// TIA Portal project "final" (V16)

(* hardware
DEVICE "S7-1200 station_1"  S7-1200 Station
   slot 0: "Rack_0"  S7-1200 Rack  Rack  V1.0
   slot 1: "PLC_1"  CPU 1212C AC/DC/Rly  6ES7 212-1BE40-0XB0  V4.0
*)

// ===== PLC "PLC_1"  CPU 1212C AC/DC/Rly =====

VAR_GLOBAL   // PLC tag table "Default tag table"
   "Tag_1" AT %I0.7 : Bool;
   "Tag_2" AT %Q0.5 : Bool;
   "Tag_3" AT %M0.0 : Bool;
   "Tag_4" AT %M1.1 : Bool;
   "Tag_5" AT %M1.2 : Bool;
   "Tag_6" AT %M2.1 : Bool;
   "Tag_7" AT %Q0.3 : Bool;
   "Tag_8" AT %M0.1 : Bool;
   "Tag_9" AT %M1.3 : Bool;
   "Tag_10" AT %M3.1 : Bool;
   "Tag_11" AT %M0.2 : Bool;
   "Tag_12" AT %M4.1 : Bool;
   "Tag_13" AT %M3.2 : Bool;
   "Tag_14" AT %M2.2 : Bool;
   "Tag_15" AT %M0.3 : Bool;
   "Tag_16" AT %M4.2 : Bool;
   "Tag_17" AT %M3.3 : Bool;
   "Tag_18" AT %M2.3 : Bool;
   "Tag_19" AT %M0.5 : Bool;
   "Tag_20" AT %M4.3 : Bool;
   "Tag_21" AT %M0.6 : Bool;
   "Tag_22" AT %Q0.4 : Bool;
   "Tag_23" AT %Q0.2 : Bool;
END_VAR

// folder: System blocks/Program resources

DATA_BLOCK "0"   // DB1
{ S7_Optimized_Access := 'TRUE' }
AUTHOR : Simatic
FAMILY : IEC
NAME : IEC_TMR
VERSION : 1.0
// stored: InstanceOfName IEC_TIMER
"IEC_TIMER"
BEGIN
END_DATA_BLOCK

DATA_BLOCK "1"   // DB2
{ S7_Optimized_Access := 'TRUE' }
AUTHOR : Simatic
FAMILY : IEC
NAME : IEC_TMR
VERSION : 1.0
// stored: InstanceOfName IEC_TIMER
"IEC_TIMER"
BEGIN
END_DATA_BLOCK

DATA_BLOCK "2"   // DB3
{ S7_Optimized_Access := 'TRUE' }
AUTHOR : Simatic
FAMILY : IEC
NAME : IEC_TMR
VERSION : 1.0
// stored: InstanceOfName IEC_TIMER
"IEC_TIMER"
BEGIN
END_DATA_BLOCK

DATA_BLOCK "3"   // DB4
{ S7_Optimized_Access := 'TRUE' }
AUTHOR : Simatic
FAMILY : IEC
NAME : IEC_TMR
VERSION : 1.0
// stored: InstanceOfName IEC_TIMER
"IEC_TIMER"
BEGIN
END_DATA_BLOCK

DATA_BLOCK "4"   // DB5
{ S7_Optimized_Access := 'TRUE' }
AUTHOR : Simatic
FAMILY : IEC
NAME : IEC_TMR
VERSION : 1.0
// stored: InstanceOfName IEC_TIMER
"IEC_TIMER"
BEGIN
END_DATA_BLOCK

// folder: (top level)

ORGANIZATION_BLOCK "Main"   // OB1, LAD, ProgramCycle
TITLE = "Main Program Sweep (Cycle)"
{ S7_Optimized_Access := 'TRUE' }
VERSION : 0.1
   VAR_INPUT
      Initial_Call : Bool;   // Initial call of this OB
      Remanence : Bool;   // =True, if remanent data are available
   END_VAR
   VAR_TEMP   // added for the SCL form of the ladder/FBD networks
      _w1 : Bool;
   END_VAR
BEGIN

REGION Network 1
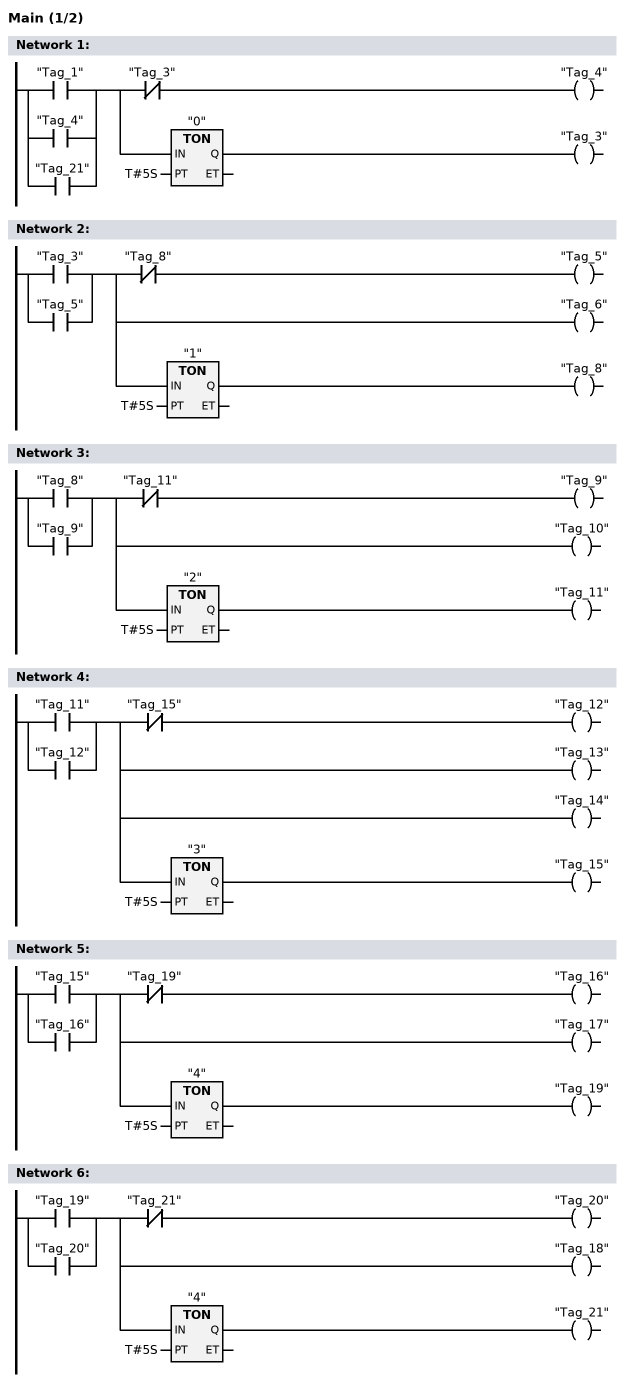
   #_w1 := "Tag_1" OR "Tag_4" OR "Tag_21";
   "Tag_4" := #_w1 AND NOT "Tag_3";
   "0".TON(IN := #_w1, PT := T#5S);
   "Tag_3" := "0".Q;
END_REGION

REGION Network 2
   #_w1 := "Tag_3" OR "Tag_5";
   "Tag_5" := #_w1 AND NOT "Tag_8";
   "Tag_6" := #_w1;
   "1".TON(IN := #_w1, PT := T#5S);
   "Tag_8" := "1".Q;
END_REGION

REGION Network 3
   #_w1 := "Tag_8" OR "Tag_9";
   "Tag_9" := #_w1 AND NOT "Tag_11";
   "Tag_10" := #_w1;
   "2".TON(IN := #_w1, PT := T#5S);
   "Tag_11" := "2".Q;
END_REGION

REGION Network 4
   #_w1 := "Tag_11" OR "Tag_12";
   "Tag_12" := #_w1 AND NOT "Tag_15";
   "Tag_13" := #_w1;
   "Tag_14" := #_w1;
   "3".TON(IN := #_w1, PT := T#5S);
   "Tag_15" := "3".Q;
END_REGION

REGION Network 5
   #_w1 := "Tag_15" OR "Tag_16";
   "Tag_16" := #_w1 AND NOT "Tag_19";
   "Tag_17" := #_w1;
   "4".TON(IN := #_w1, PT := T#5S);
   "Tag_19" := "4".Q;
END_REGION

REGION Network 6
   #_w1 := "Tag_19" OR "Tag_20";
   "Tag_20" := #_w1 AND NOT "Tag_21";
   "Tag_18" := #_w1;
   "4".TON(IN := #_w1, PT := T#5S);
   "Tag_21" := "4".Q;
END_REGION

REGION Network 7
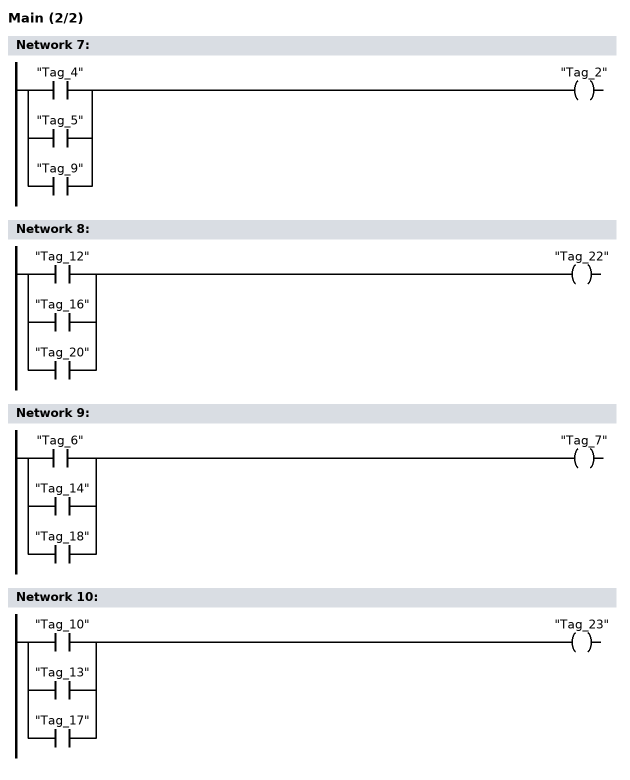
   RUNG wire#powerrail
      Contact( "Tag_4" )
      wire#w1
      Coil( "Tag_2" )
   END_RUNG
   RUNG wire#powerrail
      Contact( "Tag_5" )
   END_RUNG wire#w1
   RUNG wire#powerrail
      Contact( "Tag_9" )
   END_RUNG wire#w1
   // the same network as SCL:
   "Tag_2" := "Tag_4" OR "Tag_5" OR "Tag_9";
END_REGION

REGION Network 8
   RUNG wire#powerrail
      Contact( "Tag_12" )
      wire#w1
      Coil( "Tag_22" )
   END_RUNG
   RUNG wire#powerrail
      Contact( "Tag_16" )
   END_RUNG wire#w1
   RUNG wire#powerrail
      Contact( "Tag_20" )
   END_RUNG wire#w1
   // the same network as SCL:
   "Tag_22" := "Tag_12" OR "Tag_16" OR "Tag_20";
END_REGION

REGION Network 9
   RUNG wire#powerrail
      Contact( "Tag_6" )
      wire#w1
      Coil( "Tag_7" )
   END_RUNG
   RUNG wire#powerrail
      Contact( "Tag_14" )
   END_RUNG wire#w1
   RUNG wire#powerrail
      Contact( "Tag_18" )
   END_RUNG wire#w1
   // the same network as SCL:
   "Tag_7" := "Tag_6" OR "Tag_14" OR "Tag_18";
END_REGION

REGION Network 10
   RUNG wire#powerrail
      Contact( "Tag_10" )
      wire#w1
      Coil( "Tag_23" )
   END_RUNG
   RUNG wire#powerrail
      Contact( "Tag_13" )
   END_RUNG wire#w1
   RUNG wire#powerrail
      Contact( "Tag_17" )
   END_RUNG wire#w1
   // the same network as SCL:
   "Tag_23" := "Tag_10" OR "Tag_13" OR "Tag_17";
END_REGION
END_ORGANIZATION_BLOCK